Universal Robots URScript: movep02.script

# movep:
# Set tcp: Ignore active tcp
# Tool speed : 250mm/s
# Tool acceleration : 1200mm/s2
# Blend with radius: 25mm
# waypoint1: feature view, xyz-RxRyRz (radian), Joint positions (degree)
# Use shared blend radius
# use shared parameters

def unnamed():
  global _hidden_verificationVariable=0
  step_count_b94542ca_e842_4d6f_bfcf_1b7f83dc99ea = 0.0
  thread Step_Counter_Thread_838c19c3_aeb3_4274_b8c6_0d0273e2b71d():
    while (True):
      step_count_b94542ca_e842_4d6f_bfcf_1b7f83dc99ea = step_count_b94542ca_e842_4d6f_bfcf_1b7f83dc99ea + 1.0
      sync()
    end
  end
  run Step_Counter_Thread_838c19c3_aeb3_4274_b8c6_0d0273e2b71d()
  set_tcp(p[0.0,0.0,0.0,0.0,0.0,0.0])
  set_safety_mode_transition_hardness(1)
  set_standard_analog_input_domain(0, 1)
  set_standard_analog_input_domain(1, 1)
  set_tool_analog_input_domain(0, 1)
  set_tool_analog_input_domain(1, 1)
  set_analog_outputdomain(0, 0)
  set_analog_outputdomain(1, 0)
  set_input_actions_to_default()
  set_tool_communication(False, 115200, 0, 1, 1.5, 3.5)
  set_tool_output_mode(0)
  set_tool_digital_output_mode(0, 1)
  set_tool_digital_output_mode(1, 1)
  set_tool_voltage(0)
  set_target_payload(1.000000, [0.000000, 0.000000, 0.000000], [0.001539, 0.001539, 0.001539, 0.000000, 0.000000, 0.000000])
  set_gravity([0.0, 0.0, 9.82])
  global Waypoint_1_p=p[-.136861537556, -.267180821738, .146971261118, -.001221359682, 3.116276528482, .038891915637]
  global Waypoint_1_q=[-1.6006999999999998, -1.7271, -2.2029999999999994, -0.8079999999999998, 1.5951, -0.030999999999999694]
  while (True):
    $ 1 "Robot Program"
    $ 2 "MoveP"
    $ 3 "Waypoint_1" "breakAfter"
    movep(pose_trans(Waypoint_1_p, get_tcp_offset()), a=1.2, v=0.25, r=0.025)
  end
end
